FUNCTION WithinTolerance : BOOL
VAR_INPUT
	v1 : LREAL;
	v2 : LREAL;
	tolerance : LREAL;
END_VAR

WithinTolerance := ABS(v1-v2) < tolerance;

END_FUNCTION

(* stored: Version 1.1.0.1, ProductVersion 3.1.4024.11
   POU WithinTolerance: Id {d8380654-0700-4db5-88d4-460b84146b89}, SpecialFunc None *)
